PROGRAM MAIN
VAR
END_VAR

END_PROGRAM

(* stored: Version 1.1.0.1
   POU MAIN: Id {f7b8b195-55b7-4b22-98a4-3a9b9a6a71c6} *)
